# EPICS autosave request: ADRIXSCam/rixscamApp/Db/xcamCamera_settings.req
$(P)$(R)SEQ_FILENAME
file "RIXSCam.req", P=$(P), R=$(R)
file "ADBase_settings.req", P=$(P), R=$(R)
